// Mitsubishi GX Works2 project: 0710-온습도   PLC: Q02/Q02H

PROGRAM MAIN
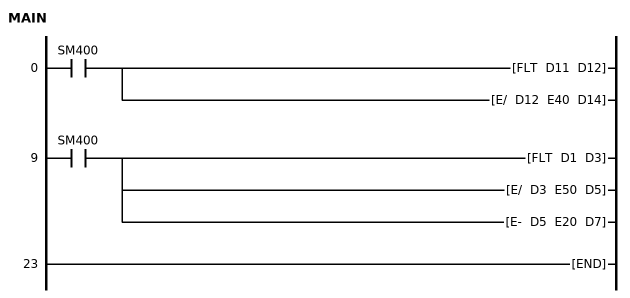
0     LD      SM400
      FLT     D11 D12
      E/      D12 E40 D14
9     LD      SM400
      FLT     D1 D3
      E/      D3 E50 D5
      E-      D5 E20 D7
23    END
END_PROGRAM
